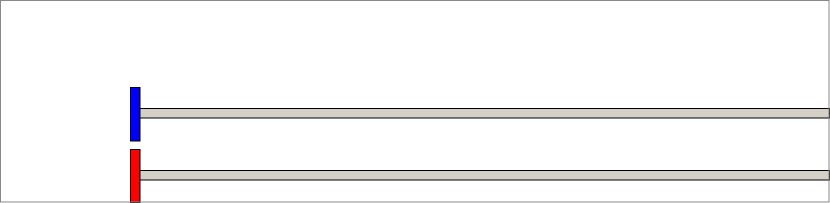
VISUALIZATION Visualization  // 830x203
    Rectangle (130,108 700x10)
    Rectangle (130,87 10x54)
        p3560616238: GVL.Achse1_Ref.NcToPlc.ActPos
    Rectangle (130,170 700x10)
    Rectangle (130,149 10x54)
        p3560616238: GVL.Achse2_Ref.NcToPlc.ActPos
END_VISUALIZATION

(* stored: Version 1.1.0.1, ProductVersion 3.1.4024.4
   Visu Visualization: Id {8dabf14e-0b9e-4b40-81d6-e0d327bd5860} *)
